// Mitsubishi GX Works2 project: 安藤間北西線FLEX   PLC: Q02/Q02H

PROGRAM FLEXPIWI  // PID演算 for WIndows
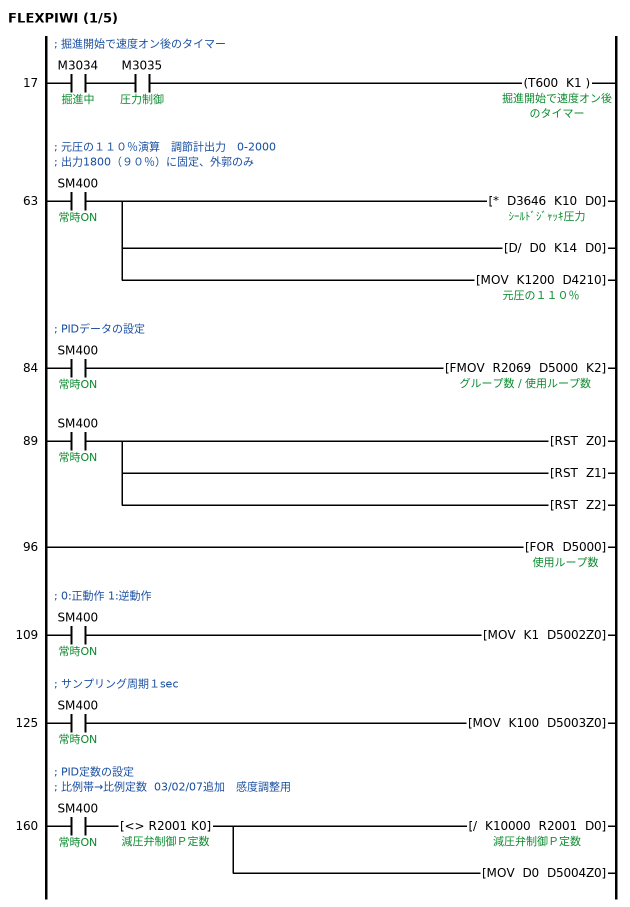
; 掘進開始で速度オン後のタイマー
17    LD      M3034  ; 掘進中
      AND     M3035  ; 圧力制御
      OUT     T600 K1  ; 掘進開始で速度オン後のタイマー
; 元圧の１１０％演算　調節計出力　0-2000
; 出力1800（９０％）に固定、外郭のみ
63    LD      SM400  ; 常時ON
      *       D3646 K10 D0  ; ｼｰﾙﾄﾞｼﾞｬｯｷ圧力
      D/      D0 K14 D0
      MOV     K1200 D4210  ; 元圧の１１０％
; PIDデータの設定
84    LD      SM400  ; 常時ON
      FMOV    R2069 D5000 K2  ; グループ数 / 使用ループ数
89    LD      SM400  ; 常時ON
      RST     Z0
      RST     Z1
      RST     Z2
96    FOR     D5000
; 0:正動作 1:逆動作
109   LD      SM400  ; 常時ON
      MOV     K1 D5002Z0
; サンプリング周期１sec
125   LD      SM400  ; 常時ON
      MOV     K100 D5003Z0
; PID定数の設定
; 比例帯→比例定数  03/02/07追加　感度調整用
160   LD      SM400  ; 常時ON
      AND<>   R2001 K0  ; 減圧弁制御Ｐ定数
      /       K10000 R2001 D0
      MOV     D0 D5004Z0
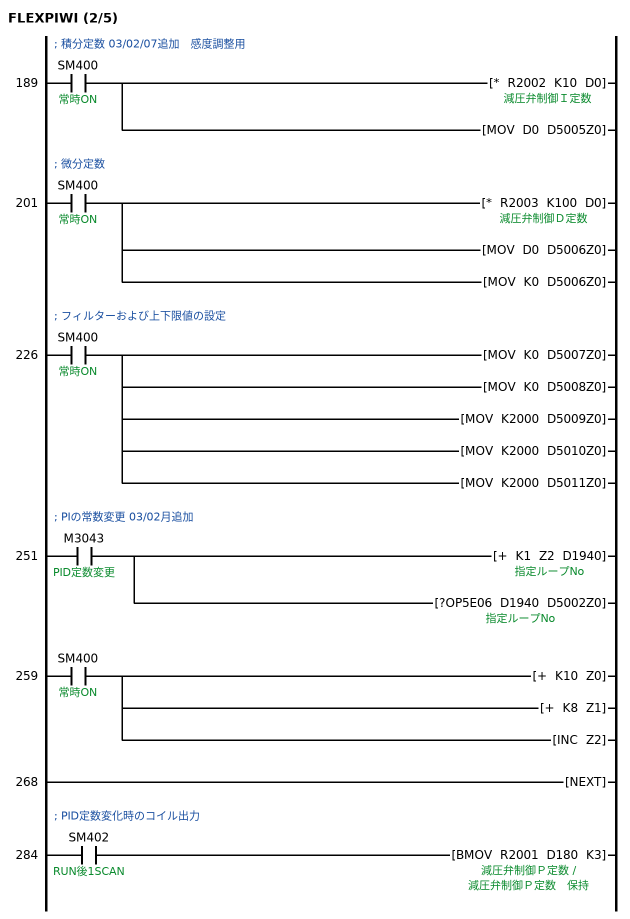
; 積分定数 03/02/07追加　感度調整用
189   LD      SM400  ; 常時ON
      *       R2002 K10 D0  ; 減圧弁制御Ｉ定数
      MOV     D0 D5005Z0
; 微分定数
201   LD      SM400  ; 常時ON
      *       R2003 K100 D0  ; 減圧弁制御Ｄ定数
      MOV     D0 D5006Z0
      MOV     K0 D5006Z0
; フィルターおよび上下限値の設定
226   LD      SM400  ; 常時ON
      MOV     K0 D5007Z0
      MOV     K0 D5008Z0
      MOV     K2000 D5009Z0
      MOV     K2000 D5010Z0
      MOV     K2000 D5011Z0
; PIの常数変更 03/02月追加
251   LD      M3043  ; PID定数変更
      +       K1 Z2 D1940  ; 指定ループNo
      ?OP5E06 D1940 D5002Z0
259   LD      SM400  ; 常時ON
      +       K10 Z0
      +       K8 Z1
      INC     Z2
268   NEXT
; PID定数変化時のコイル出力
284   LD      SM402  ; RUN後1SCAN
      BMOV    R2001 D180 K3  ; 減圧弁制御Ｐ定数　保持
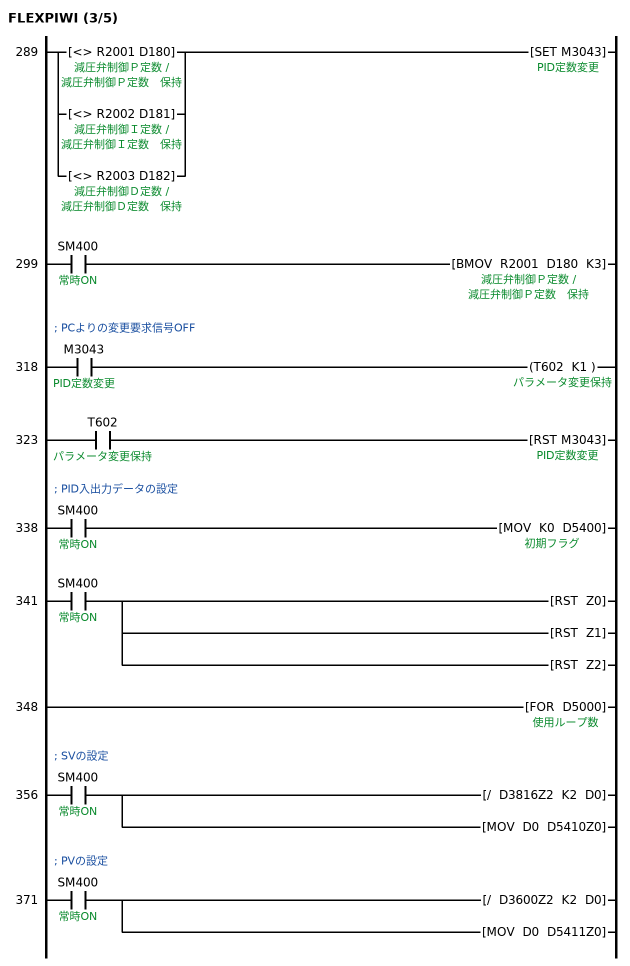
289   LD<>    R2001 D180  ; 減圧弁制御Ｐ定数 / 減圧弁制御Ｐ定数　保持
      OR<>    R2002 D181  ; 減圧弁制御Ｉ定数 / 減圧弁制御Ｉ定数　保持
      OR<>    R2003 D182  ; 減圧弁制御Ｄ定数 / 減圧弁制御Ｄ定数　保持
      SET     M3043  ; PID定数変更
299   LD      SM400  ; 常時ON
      BMOV    R2001 D180 K3
; PCよりの変更要求信号OFF
318   LD      M3043  ; PID定数変更
      OUT     T602 K1  ; パラメータ変更保持
323   LD      T602  ; パラメータ変更保持
      RST     M3043  ; PID定数変更
; PID入出力データの設定
338   LD      SM400  ; 常時ON
      MOV     K0 D5400  ; 初期フラグ
341   LD      SM400  ; 常時ON
      RST     Z0
      RST     Z1
      RST     Z2
348   FOR     D5000
; SVの設定
356   LD      SM400  ; 常時ON
      /       D3816Z2 K2 D0
      MOV     D0 D5410Z0
; 
; PVの設定
371   LD      SM400  ; 常時ON
      /       D3600Z2 K2 D0
      MOV     D0 D5411Z0
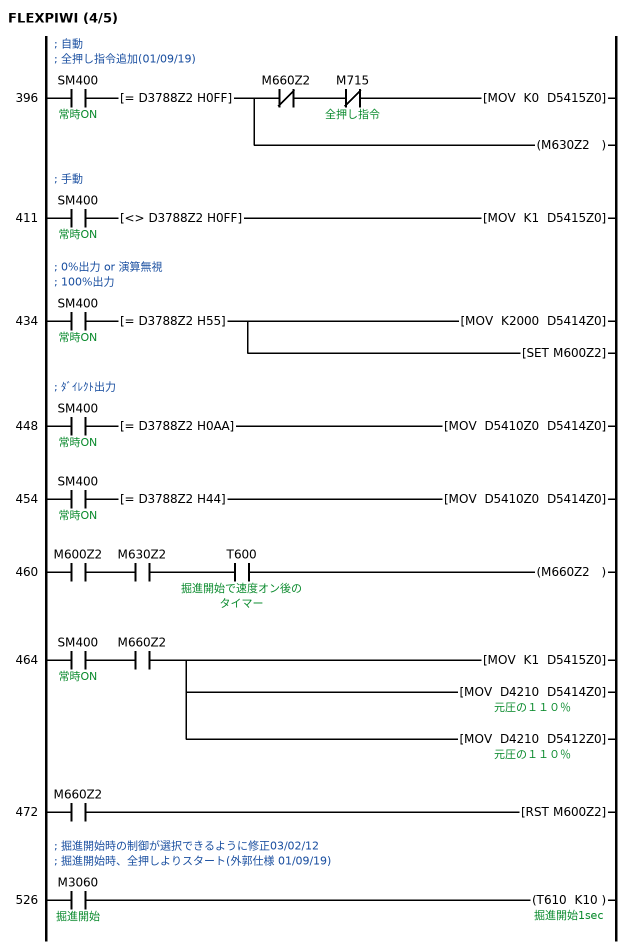
; 自動
; 全押し指令追加(01/09/19)
396   LD      SM400  ; 常時ON
      AND=    D3788Z2 H0FF
      MPS
      ANI     M660Z2
      ANI     M715  ; 全押し指令
      MOV     K0 D5415Z0
      MPP
      OUT     M630Z2
; 手動
411   LD      SM400  ; 常時ON
      AND<>   D3788Z2 H0FF
      MOV     K1 D5415Z0
; 0%出力 or 演算無視
; 100%出力
434   LD      SM400  ; 常時ON
      AND=    D3788Z2 H55
      MOV     K2000 D5414Z0
      SET     M600Z2
; ﾀﾞｲﾚｸﾄ出力
448   LD      SM400  ; 常時ON
      AND=    D3788Z2 H0AA
      MOV     D5410Z0 D5414Z0
454   LD      SM400  ; 常時ON
      AND=    D3788Z2 H44
      MOV     D5410Z0 D5414Z0
460   LD      M600Z2
      AND     M630Z2
      AND     T600  ; 掘進開始で速度オン後のタイマー
      OUT     M660Z2
464   LD      SM400  ; 常時ON
      AND     M660Z2
      MOV     K1 D5415Z0
      MOV     D4210 D5414Z0
      MOV     D4210 D5412Z0
472   LD      M660Z2
      RST     M600Z2
; 掘進開始時の制御が選択できるように修正03/02/12
; 掘進開始時、全押しよりスタート(外郭仕様 01/09/19)
526   LD      M3060  ; 掘進開始
      OUT     T610 K10  ; 掘進開始1sec
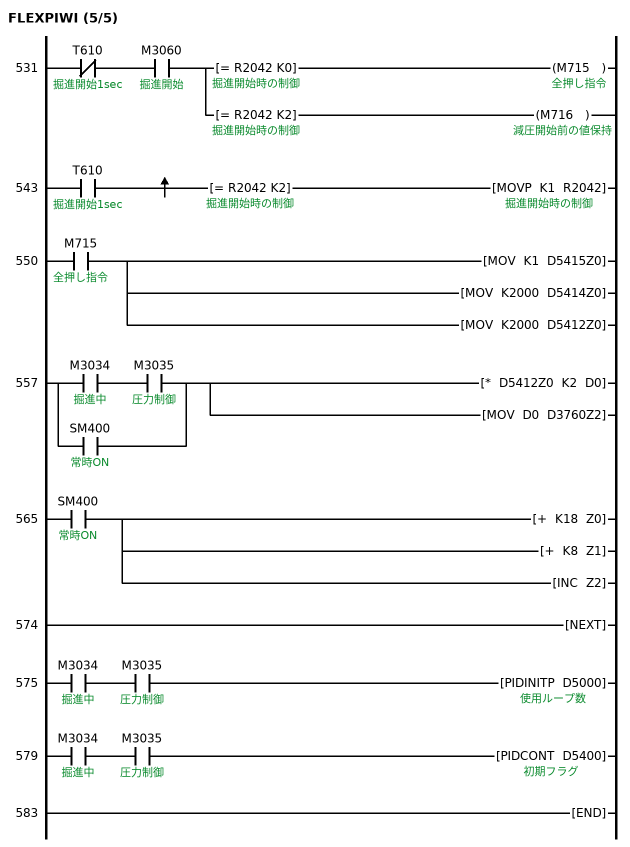
531   LDI     T610  ; 掘進開始1sec
      AND     M3060  ; 掘進開始
      MPS
      AND=    R2042 K0  ; 掘進開始時の制御
      OUT     M715  ; 全押し指令
      MPP
      AND=    R2042 K2  ; 掘進開始時の制御
      OUT     M716  ; 減圧開始前の値保持
543   LD      T610  ; 掘進開始1sec
      MEP
      AND=    R2042 K2  ; 掘進開始時の制御
      MOVP    K1 R2042
550   LD      M715  ; 全押し指令
      MOV     K1 D5415Z0
      MOV     K2000 D5414Z0
      MOV     K2000 D5412Z0
557   LD      M3034  ; 掘進中
      AND     M3035  ; 圧力制御
      OR      SM400  ; 常時ON
      *       D5412Z0 K2 D0
      MOV     D0 D3760Z2
565   LD      SM400  ; 常時ON
      +       K18 Z0
      +       K8 Z1
      INC     Z2
574   NEXT
575   LD      M3034  ; 掘進中
      AND     M3035  ; 圧力制御
      PIDINITP D5000
579   LD      M3034  ; 掘進中
      AND     M3035  ; 圧力制御
      PIDCONT D5400
583   END
END_PROGRAM

PROGRAM FLEXWIN  // FlexWindos対応
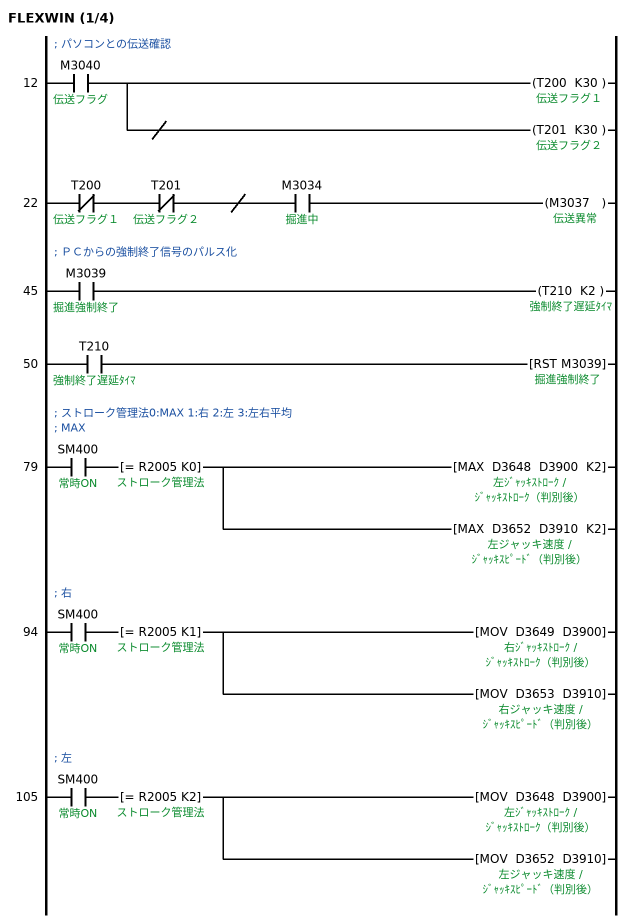
; パソコンとの伝送確認
12    LD      M3040  ; 伝送フラグ
      OUT     T200 K30  ; 伝送フラグ１
      INV
      OUT     T201 K30  ; 伝送フラグ２
22    LDI     T200  ; 伝送フラグ１
      ANI     T201  ; 伝送フラグ２
      INV
      AND     M3034  ; 掘進中
      OUT     M3037  ; 伝送異常
; ＰＣからの強制終了信号のパルス化
45    LD      M3039  ; 掘進強制終了
      OUT     T210 K2  ; 強制終了遅延ﾀｲﾏ
50    LD      T210  ; 強制終了遅延ﾀｲﾏ
      RST     M3039  ; 掘進強制終了
; ストローク管理法0:MAX 1:右 2:左 3:左右平均
; MAX
79    LD      SM400  ; 常時ON
      AND=    R2005 K0  ; ストローク管理法
      MAX     D3648 D3900 K2  ; 左ｼﾞｬｯｷｽﾄﾛｰｸ / ｼﾞｬｯｷｽﾄﾛｰｸ（判別後）
      MAX     D3652 D3910 K2  ; 左ジャッキ速度 / ｼﾞｬｯｷｽﾋﾟｰﾄﾞ（判別後）
; 右
94    LD      SM400  ; 常時ON
      AND=    R2005 K1  ; ストローク管理法
      MOV     D3649 D3900  ; 右ｼﾞｬｯｷｽﾄﾛｰｸ
      MOV     D3653 D3910  ; 右ジャッキ速度
; 左
105   LD      SM400  ; 常時ON
      AND=    R2005 K2  ; ストローク管理法
      MOV     D3648 D3900
      MOV     D3652 D3910
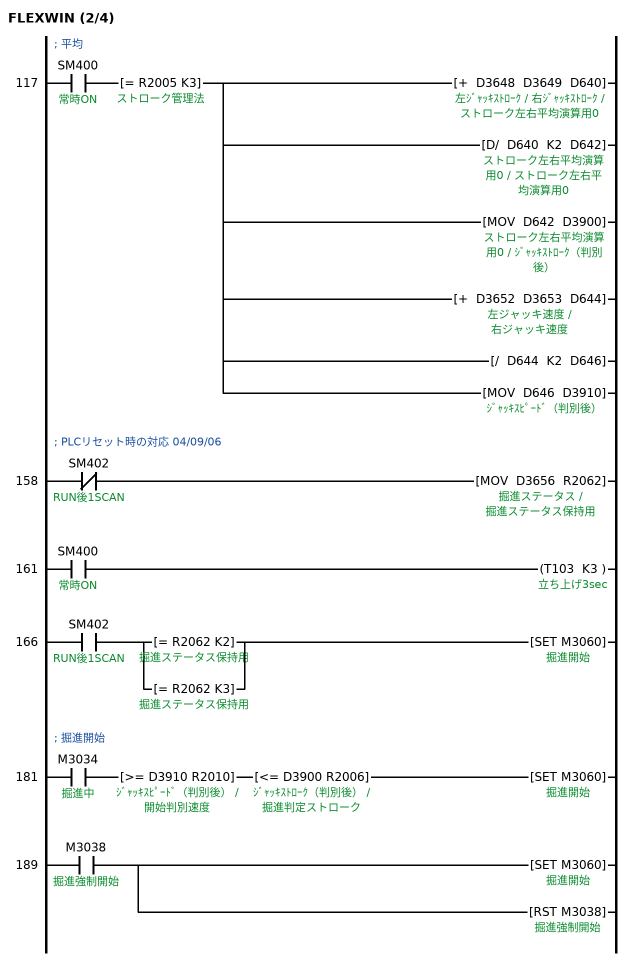
; 平均
117   LD      SM400  ; 常時ON
      AND=    R2005 K3  ; ストローク管理法
      +       D3648 D3649 D640  ; ストローク左右平均演算用0
      D/      D640 K2 D642  ; ストローク左右平均演算用0
      MOV     D642 D3900
      +       D3652 D3653 D644
      /       D644 K2 D646
      MOV     D646 D3910
; PLCリセット時の対応 04/09/06
158   LDI     SM402  ; RUN後1SCAN
      MOV     D3656 R2062  ; 掘進ステータス / 掘進ステータス保持用
161   LD      SM400  ; 常時ON
      OUT     T103 K3  ; 立ち上げ3sec
166   LD      SM402  ; RUN後1SCAN
      LD=     R2062 K2  ; 掘進ステータス保持用
      OR=     R2062 K3  ; 掘進ステータス保持用
      ANB
      SET     M3060  ; 掘進開始
; 掘進開始
181   LD      M3034  ; 掘進中
      AND>=   D3910 R2010  ; ｼﾞｬｯｷｽﾋﾟｰﾄﾞ（判別後） / 開始判別速度
      AND<=   D3900 R2006  ; ｼﾞｬｯｷｽﾄﾛｰｸ（判別後） / 掘進判定ストローク
      SET     M3060  ; 掘進開始
189   LD      M3038  ; 掘進強制開始
      SET     M3060  ; 掘進開始
      RST     M3038  ; 掘進強制開始
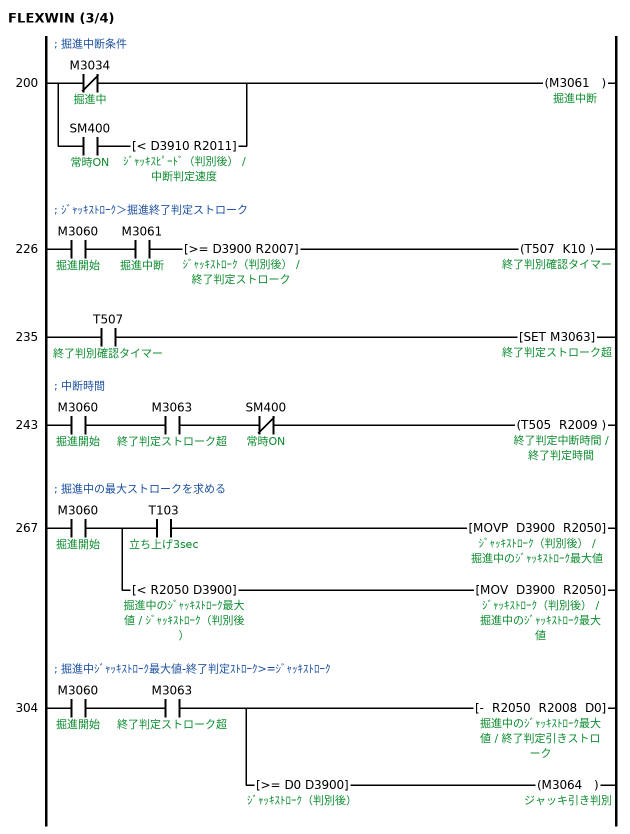
; 掘進中断条件
200   LDI     M3034  ; 掘進中
      LD      SM400  ; 常時ON
      AND<    D3910 R2011  ; ｼﾞｬｯｷｽﾋﾟｰﾄﾞ（判別後） / 中断判定速度
      ORB
      OUT     M3061  ; 掘進中断
; ｼﾞｬｯｷｽﾄﾛｰｸ＞掘進終了判定ストローク
226   LD      M3060  ; 掘進開始
      AND     M3061  ; 掘進中断
      AND>=   D3900 R2007  ; ｼﾞｬｯｷｽﾄﾛｰｸ（判別後） / 終了判定ストローク
      OUT     T507 K10  ; 終了判別確認タイマー
235   LD      T507  ; 終了判別確認タイマー
      SET     M3063  ; 終了判定ストローク超
; 中断時間
243   LD      M3060  ; 掘進開始
      AND     M3063  ; 終了判定ストローク超
      ANI     SM400  ; 常時ON
      OUT     T505 R2009  ; 終了判定中断時間 / 終了判定時間
; 掘進中の最大ストロークを求める
267   LD      M3060  ; 掘進開始
      MPS
      AND     T103  ; 立ち上げ3sec
      MOVP    D3900 R2050  ; 掘進中のｼﾞｬｯｷｽﾄﾛｰｸ最大値
      MPP
      AND<    R2050 D3900  ; 掘進中のｼﾞｬｯｷｽﾄﾛｰｸ最大値 / ｼﾞｬｯｷｽﾄﾛｰｸ（判別後）
      MOV     D3900 R2050
; 掘進中ｼﾞｬｯｷｽﾄﾛｰｸ最大値-終了判定ｽﾄﾛｰｸ>=ｼﾞｬｯｷｽﾄﾛｰｸ
304   LD      M3060  ; 掘進開始
      AND     M3063  ; 終了判定ストローク超
      -       R2050 R2008 D0  ; 終了判定引きストローク
      AND>=   D0 D3900  ; ｼﾞｬｯｷｽﾄﾛｰｸ（判別後）
      OUT     M3064  ; ジャッキ引き判別
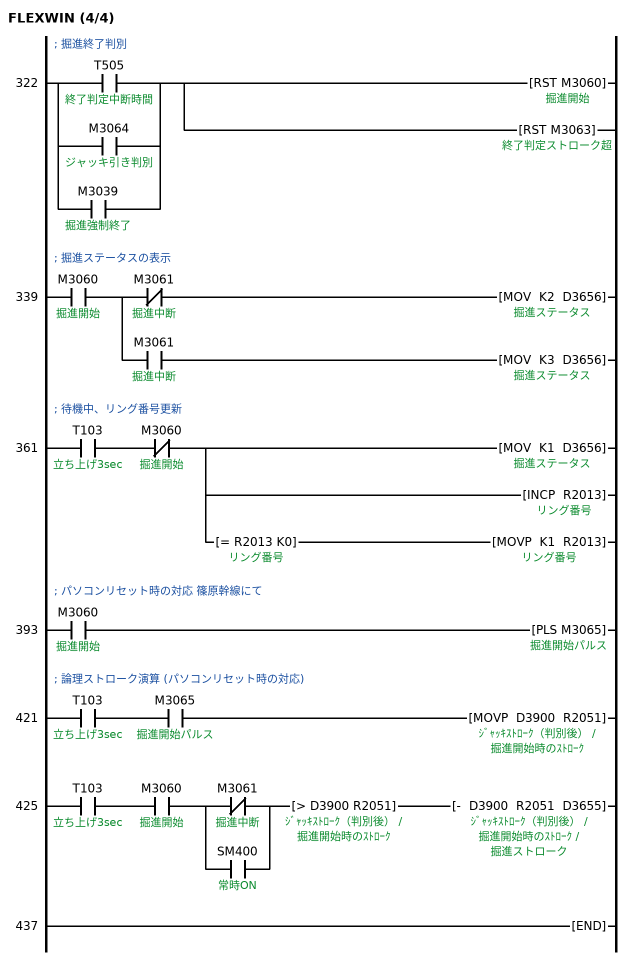
; 掘進終了判別
322   LD      T505  ; 終了判定中断時間
      OR      M3064  ; ジャッキ引き判別
      OR      M3039  ; 掘進強制終了
      RST     M3060  ; 掘進開始
      RST     M3063  ; 終了判定ストローク超
; 掘進ステータスの表示
339   LD      M3060  ; 掘進開始
      MPS
      ANI     M3061  ; 掘進中断
      MOV     K2 D3656
      MPP
      AND     M3061  ; 掘進中断
      MOV     K3 D3656
; 待機中、リング番号更新
361   LD      T103  ; 立ち上げ3sec
      ANI     M3060  ; 掘進開始
      MOV     K1 D3656
      INCP    R2013  ; リング番号
      AND=    R2013 K0  ; リング番号
      MOVP    K1 R2013
; パソコンリセット時の対応 篠原幹線にて
393   LD      M3060  ; 掘進開始
      PLS     M3065  ; 掘進開始パルス
; 論理ストローク演算 (パソコンリセット時の対応)
421   LD      T103  ; 立ち上げ3sec
      AND     M3065  ; 掘進開始パルス
      MOVP    D3900 R2051  ; 掘進開始時のｽﾄﾛｰｸ
425   LD      T103  ; 立ち上げ3sec
      AND     M3060  ; 掘進開始
      LDI     M3061  ; 掘進中断
      OR      SM400  ; 常時ON
      ANB
      AND>    D3900 R2051  ; ｼﾞｬｯｷｽﾄﾛｰｸ（判別後） / 掘進開始時のｽﾄﾛｰｸ
      -       D3900 R2051 D3655  ; 掘進ストローク
437   END
END_PROGRAM

PROGRAM INOUTWIN  // 安藤間北西線FLEX
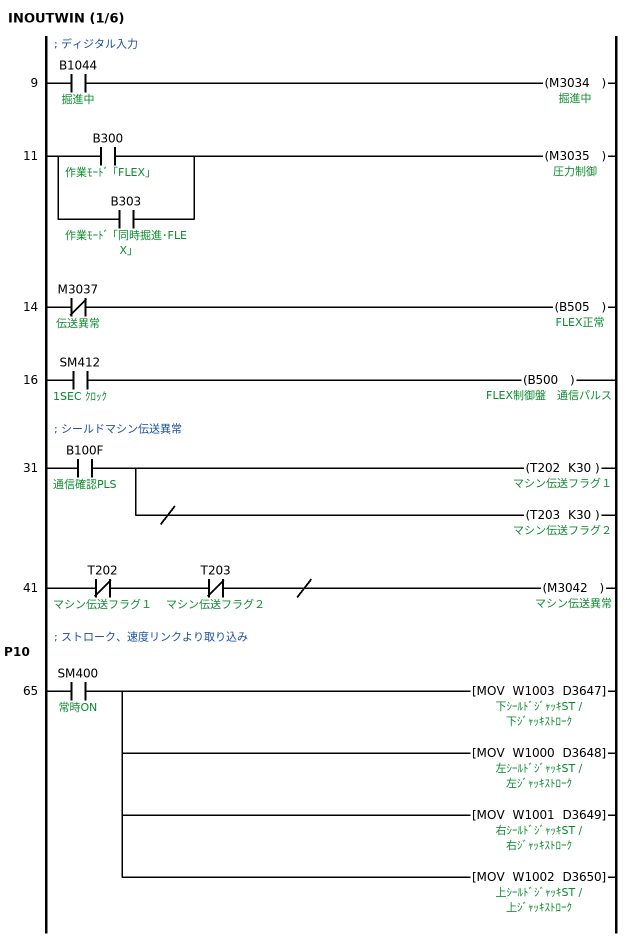
; ディジタル入力
9     LD      B1044  ; 掘進中
      OUT     M3034  ; 掘進中
11    LD      B300  ; 作業ﾓｰﾄﾞ ｢FLEX｣
      OR      B303  ; 作業ﾓｰﾄﾞ ｢同時掘進･FLEX｣
      OUT     M3035  ; 圧力制御
14    LDI     M3037  ; 伝送異常
      OUT     B505  ; FLEX正常
16    LD      SM412  ; 1SEC ｸﾛｯｸ
      OUT     B500  ; FLEX制御盤　通信パルス
; シールドマシン伝送異常
31    LD      B100F  ; 通信確認PLS
      OUT     T202 K30  ; マシン伝送フラグ１
      INV
      OUT     T203 K30  ; マシン伝送フラグ２
41    LDI     T202  ; マシン伝送フラグ１
      ANI     T203  ; マシン伝送フラグ２
      INV
      OUT     M3042  ; マシン伝送異常
; ストローク、速度リンクより取り込み
      P10
65    LD      SM400  ; 常時ON
      MOV     W1003 D3647  ; 下ｼｰﾙﾄﾞｼﾞｬｯｷST / 下ｼﾞｬｯｷｽﾄﾛｰｸ
      MOV     W1000 D3648  ; 左ｼｰﾙﾄﾞｼﾞｬｯｷST / 左ｼﾞｬｯｷｽﾄﾛｰｸ
      MOV     W1001 D3649  ; 右ｼｰﾙﾄﾞｼﾞｬｯｷST / 右ｼﾞｬｯｷｽﾄﾛｰｸ
      MOV     W1002 D3650  ; 上ｼｰﾙﾄﾞｼﾞｬｯｷST / 上ｼﾞｬｯｷｽﾄﾛｰｸ
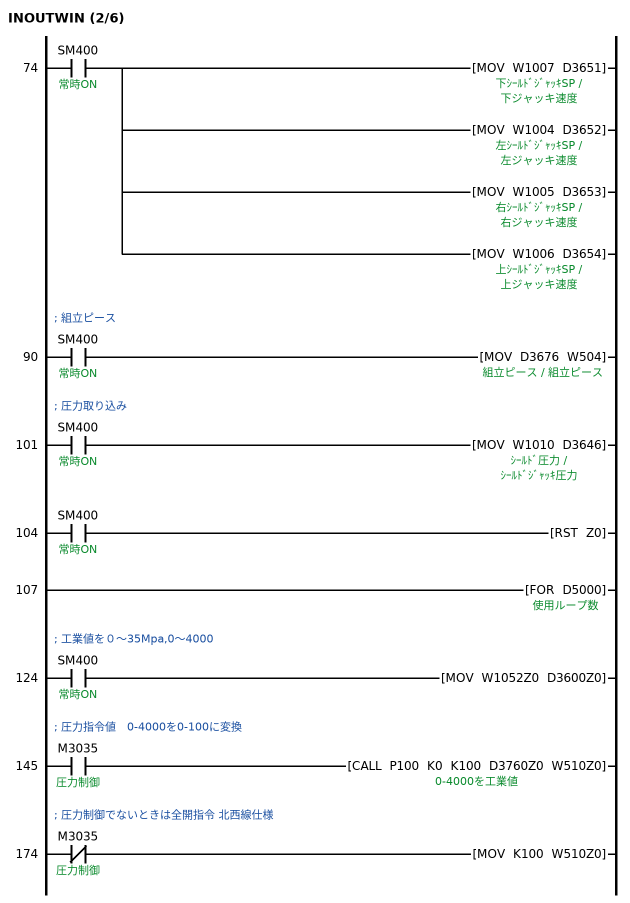
74    LD      SM400  ; 常時ON
      MOV     W1007 D3651  ; 下ｼｰﾙﾄﾞｼﾞｬｯｷSP / 下ジャッキ速度
      MOV     W1004 D3652  ; 左ｼｰﾙﾄﾞｼﾞｬｯｷSP / 左ジャッキ速度
      MOV     W1005 D3653  ; 右ｼｰﾙﾄﾞｼﾞｬｯｷSP / 右ジャッキ速度
      MOV     W1006 D3654  ; 上ｼｰﾙﾄﾞｼﾞｬｯｷSP / 上ジャッキ速度
; 組立ピース
90    LD      SM400  ; 常時ON
      MOV     D3676 W504  ; 組立ピース / 組立ピース
; 圧力取り込み
101   LD      SM400  ; 常時ON
      MOV     W1010 D3646  ; ｼｰﾙﾄﾞ圧力 / ｼｰﾙﾄﾞｼﾞｬｯｷ圧力
104   LD      SM400  ; 常時ON
      RST     Z0
107   FOR     D5000  ; 使用ループ数
; 工業値を０～35Mpa,0～4000
124   LD      SM400  ; 常時ON
      MOV     W1052Z0 D3600Z0
; 圧力指令値　0-4000を0-100に変換
145   LD      M3035  ; 圧力制御
      CALL    P100 K0 K100 D3760Z0 W510Z0  ; 0-4000を工業値
; 圧力制御でないときは全開指令 北西線仕様
174   LDI     M3035  ; 圧力制御
      MOV     K100 W510Z0
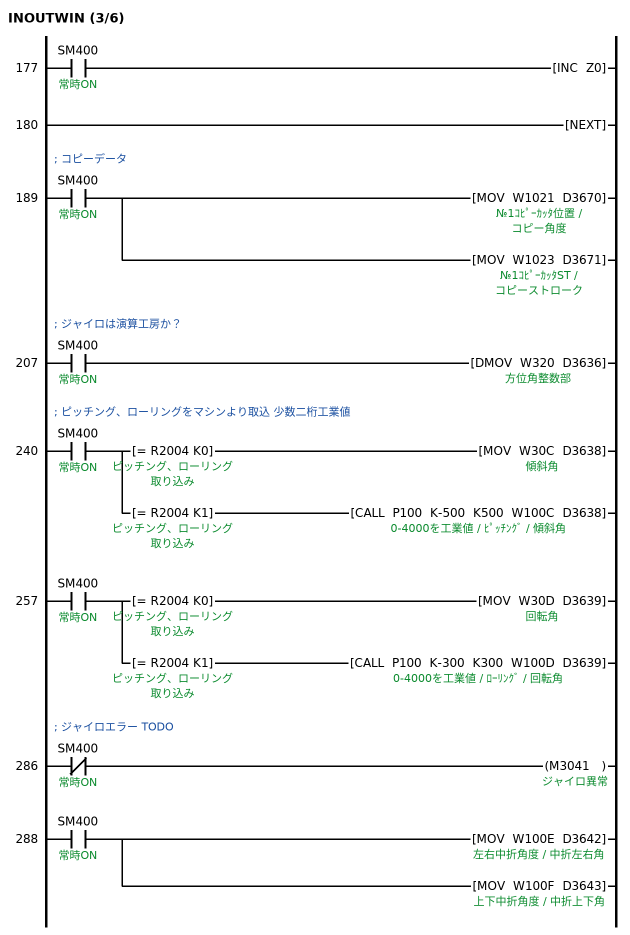
177   LD      SM400  ; 常時ON
      INC     Z0
180   NEXT
; コピーデータ
189   LD      SM400  ; 常時ON
      MOV     W1021 D3670  ; №1ｺﾋﾟｰｶｯﾀ位置 / コピー角度
      MOV     W1023 D3671  ; №1ｺﾋﾟｰｶｯﾀST / コピーストローク
; ジャイロは演算工房か？
207   LD      SM400  ; 常時ON
      DMOV    W320 D3636  ; 方位角整数部
; ピッチング、ローリングをマシンより取込 少数二桁工業値
240   LD      SM400  ; 常時ON
      MPS
      AND=    R2004 K0  ; ピッチング、ローリング取り込み
      MOV     W30C D3638  ; 傾斜角
      MPP
      AND=    R2004 K1  ; ピッチング、ローリング取り込み
      CALL    P100 K-500 K500 W100C D3638  ; ﾋﾟｯﾁﾝｸﾞ
257   LD      SM400  ; 常時ON
      MPS
      AND=    R2004 K0  ; ピッチング、ローリング取り込み
      MOV     W30D D3639  ; 回転角
      MPP
      AND=    R2004 K1  ; ピッチング、ローリング取り込み
      CALL    P100 K-300 K300 W100D D3639  ; ﾛｰﾘﾝｸﾞ
; ジャイロエラー TODO
286   LDI     SM400  ; 常時ON
      OUT     M3041  ; ジャイロ異常
288   LD      SM400  ; 常時ON
      MOV     W100E D3642  ; 左右中折角度 / 中折左右角
      MOV     W100F D3643  ; 上下中折角度 / 中折上下角
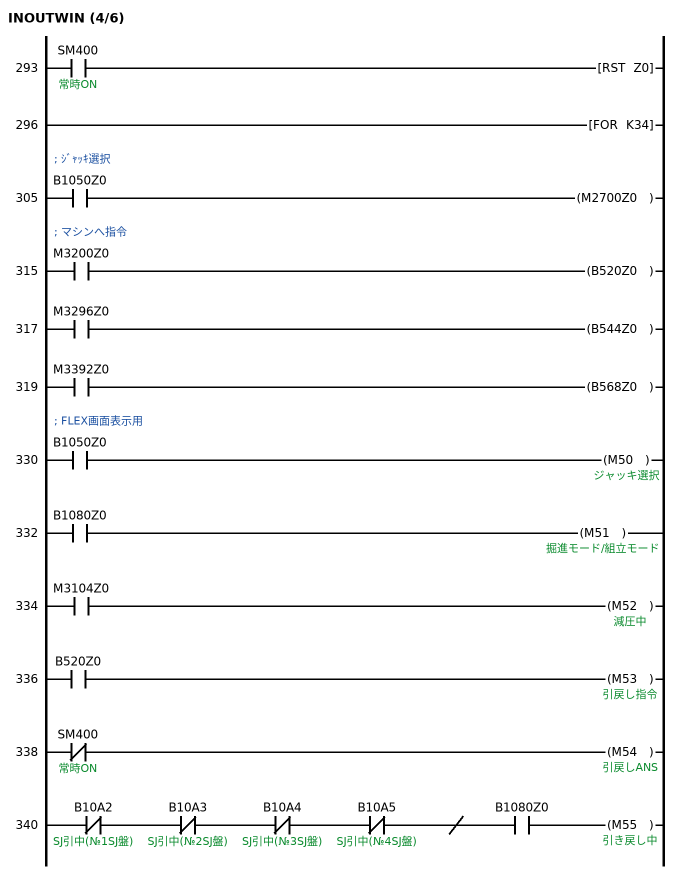
293   LD      SM400  ; 常時ON
      RST     Z0
296   FOR     K34
; ｼﾞｬｯｷ選択
305   LD      B1050Z0
      OUT     M2700Z0
; マシンへ指令
315   LD      M3200Z0
      OUT     B520Z0
317   LD      M3296Z0
      OUT     B544Z0
319   LD      M3392Z0
      OUT     B568Z0
; FLEX画面表示用
330   LD      B1050Z0
      OUT     M50  ; ジャッキ選択
332   LD      B1080Z0
      OUT     M51  ; 掘進モード/組立モード
334   LD      M3104Z0
      OUT     M52  ; 減圧中
336   LD      B520Z0
      OUT     M53  ; 引戻し指令
338   LDI     SM400  ; 常時ON
      OUT     M54  ; 引戻しANS
340   LDI     B10A2  ; SJ引中(№1SJ盤)
      ANI     B10A3  ; SJ引中(№2SJ盤)
      ANI     B10A4  ; SJ引中(№3SJ盤)
      ANI     B10A5  ; SJ引中(№4SJ盤)
      INV
      AND     B1080Z0
      OUT     M55  ; 引き戻し中
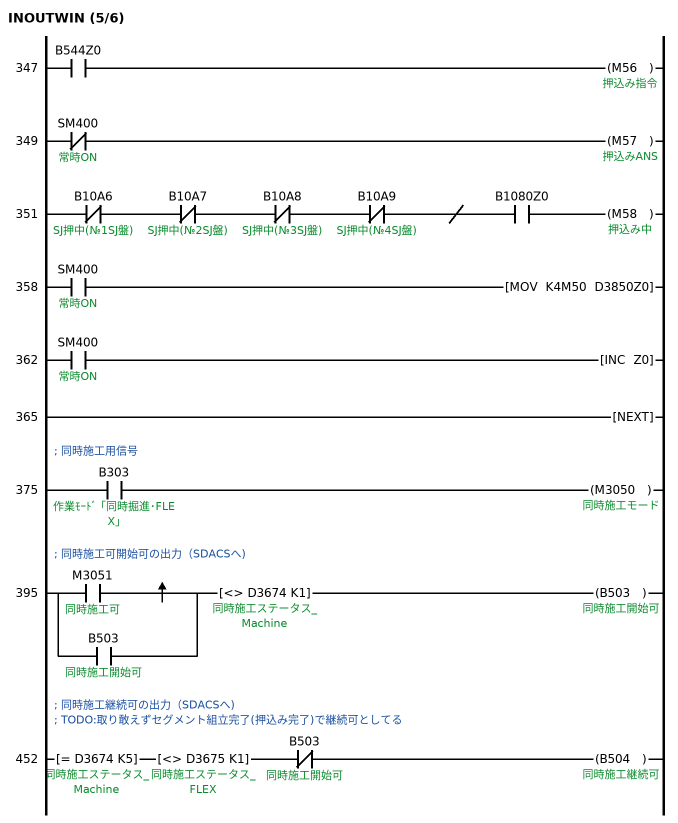
347   LD      B544Z0
      OUT     M56  ; 押込み指令
349   LDI     SM400  ; 常時ON
      OUT     M57  ; 押込みANS
351   LDI     B10A6  ; SJ押中(№1SJ盤)
      ANI     B10A7  ; SJ押中(№2SJ盤)
      ANI     B10A8  ; SJ押中(№3SJ盤)
      ANI     B10A9  ; SJ押中(№4SJ盤)
      INV
      AND     B1080Z0
      OUT     M58  ; 押込み中
358   LD      SM400  ; 常時ON
      MOV     K4M50 D3850Z0
362   LD      SM400  ; 常時ON
      INC     Z0
365   NEXT
; 同時施工用信号
375   LD      B303  ; 作業ﾓｰﾄﾞ ｢同時掘進･FLEX｣
      OUT     M3050  ; 同時施工モード
; 同時施工可開始可の出力（SDACSへ)
395   LD      M3051  ; 同時施工可
      MEP
      OR      B503  ; 同時施工開始可
      AND<>   D3674 K1  ; 同時施工ステータス_Machine
      OUT     B503  ; 同時施工開始可
; 同時施工継続可の出力（SDACSへ)
; TODO:取り敢えずセグメント組立完了(押込み完了)で継続可としてる
452   LD=     D3674 K5  ; 同時施工ステータス_Machine
      AND<>   D3675 K1  ; 同時施工ステータス_FLEX
      ANI     B503  ; 同時施工開始可
      OUT     B504  ; 同時施工継続可
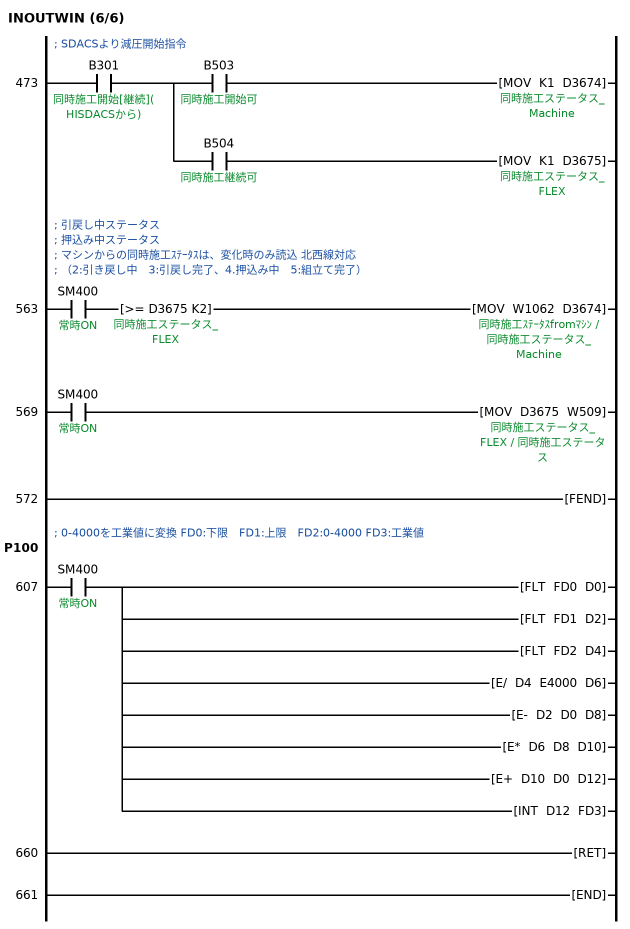
; SDACSより減圧開始指令
473   LD      B301  ; 同時施工開始[継続](HISDACSから)
      MPS
      AND     B503  ; 同時施工開始可
      MOV     K1 D3674
      MPP
      AND     B504  ; 同時施工継続可
      MOV     K1 D3675
; 引戻し中ステータス
; 押込み中ステータス
; マシンからの同時施工ｽﾃｰﾀｽは、変化時のみ読込 北西線対応
; （2:引き戻し中　3:引戻し完了、4.押込み中　5:組立て完了）
563   LD      SM400  ; 常時ON
      AND>=   D3675 K2  ; 同時施工ステータス_FLEX
      MOV     W1062 D3674  ; 同時施工ｽﾃｰﾀｽfromﾏｼﾝ
569   LD      SM400  ; 常時ON
      MOV     D3675 W509  ; 同時施工ステータス
572   FEND
      P100
; 0-4000を工業値に変換 FD0:下限　FD1:上限　FD2:0-4000 FD3:工業値
607   LD      SM400  ; 常時ON
      FLT     FD0 D0
        [note] スケール上限
      FLT     FD1 D2
        [note] スケール下限
      FLT     FD2 D4
        [note] 元アドレス
      E/      D4 E4000 D6
      E-      D2 D0 D8
      E*      D6 D8 D10
      E+      D10 D0 D12
      INT     D12 FD3
660   RET
661   END
END_PROGRAM

PROGRAM Simlat  // 安藤間北西線シュミレーション
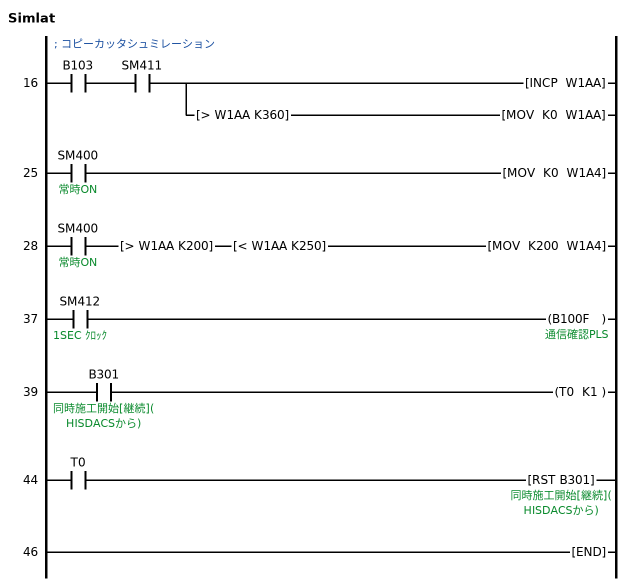
; コピーカッタシュミレーション
16    LD      B103
      AND     SM411
      INCP    W1AA
      AND>    W1AA K360
      MOV     K0 W1AA
25    LD      SM400  ; 常時ON
      MOV     K0 W1A4
28    LD      SM400  ; 常時ON
      AND>    W1AA K200
      AND<    W1AA K250
      MOV     K200 W1A4
37    LD      SM412  ; 1SEC ｸﾛｯｸ
      OUT     B100F  ; 通信確認PLS
39    LD      B301  ; 同時施工開始[継続](HISDACSから)
      OUT     T0 K1
44    LD      T0
      RST     B301  ; 同時施工開始[継続](HISDACSから)
46    END
END_PROGRAM

// device comments not shown above
D3600  ; グループ1圧力
D3816  ; グループ1圧力SV
D5002  ; グループ1演算式選択
D5412  ; グループ1自動操作量（MV)
